% RSLogix 500 project PROJECT3.RSS, saved by version 8.40.00.08 %
PROJECT "UNTITLED"    % processor: Bul.1763 MicroLogix 1100 Series B %

PROGRAM FILES
  LAD 2   22 rungs

DATA FILES
  O0 OUTPUT  4 elements
  I1 INPUT  6 elements
  S2 STATUS  66 elements
  B3 BINARY  3 elements
  T4 TIMER  1 elements
  C5 COUNTER  1 elements
  R6 CONTROL  1 elements
  N7 INTEGER  18 elements
  F8 FLOAT  1 elements
  ST9   14 elements

LADDER 2
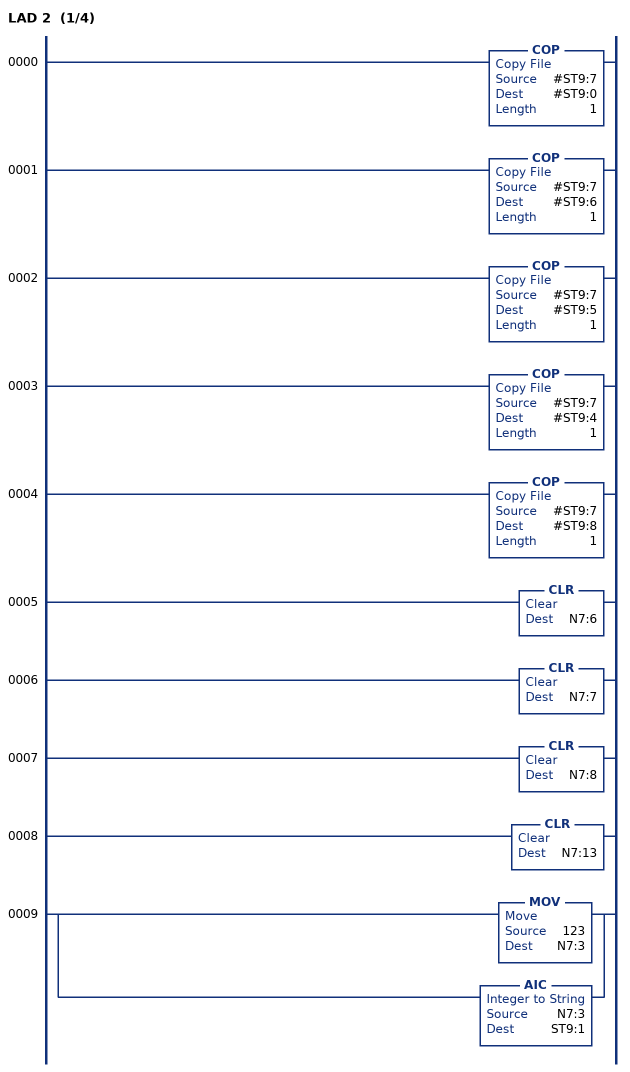
% Rung: 0 %
SOR COP #ST9:7 #ST9:0 1 EOR
% Rung: 1 %
SOR COP #ST9:7 #ST9:6 1 EOR
% Rung: 2 %
SOR COP #ST9:7 #ST9:5 1 EOR
% Rung: 3 %
SOR COP #ST9:7 #ST9:4 1 EOR
% Rung: 4 %
SOR COP #ST9:7 #ST9:8 1 EOR
% Rung: 5 %
SOR CLR N7:6 EOR
% Rung: 6 %
SOR CLR N7:7 EOR
% Rung: 7 %
SOR CLR N7:8 EOR
% Rung: 8 %
SOR CLR N7:13 EOR
% Rung: 9 %
SOR BST MOV 123 N7:3 NXB AIC N7:3 ST9:1 BND EOR

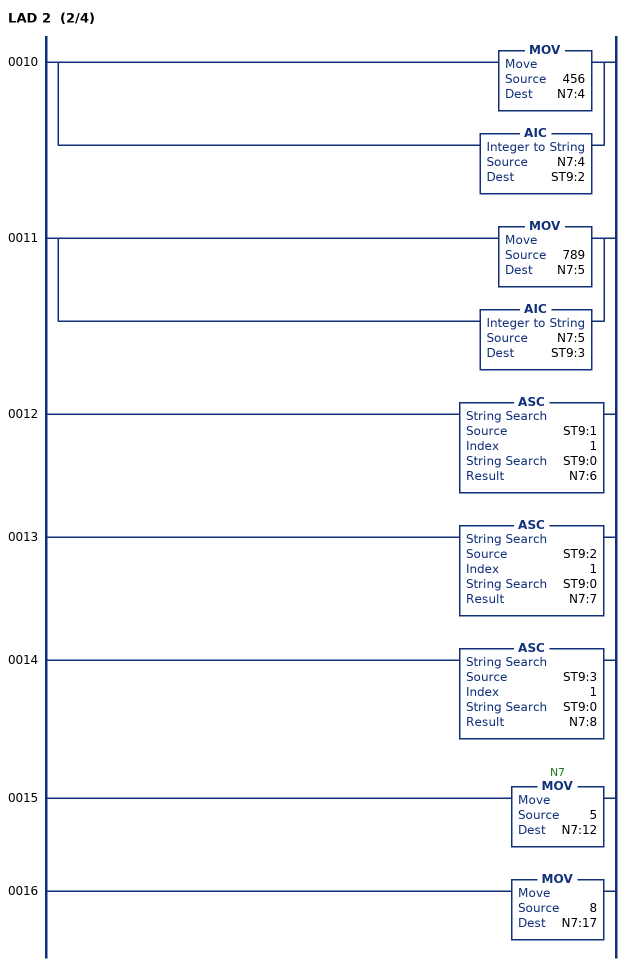
% Rung: 10 %
SOR BST MOV 456 N7:4 NXB AIC N7:4 ST9:2 BND EOR
% Rung: 11 %
SOR BST MOV 789 N7:5 NXB AIC N7:5 ST9:3 BND EOR
% Rung: 12 %
SOR ASC ST9:1 1 ST9:0 N7:6 EOR
% Rung: 13 %
SOR ASC ST9:2 1 ST9:0 N7:7 EOR
% Rung: 14 %
SOR ASC ST9:3 1 ST9:0 N7:8 EOR
% Rung: 15 %
SOR MOV 5 N7:12 EOR
%   N7:12  N7 %
% Rung: 16 %
SOR MOV 8 N7:17 EOR

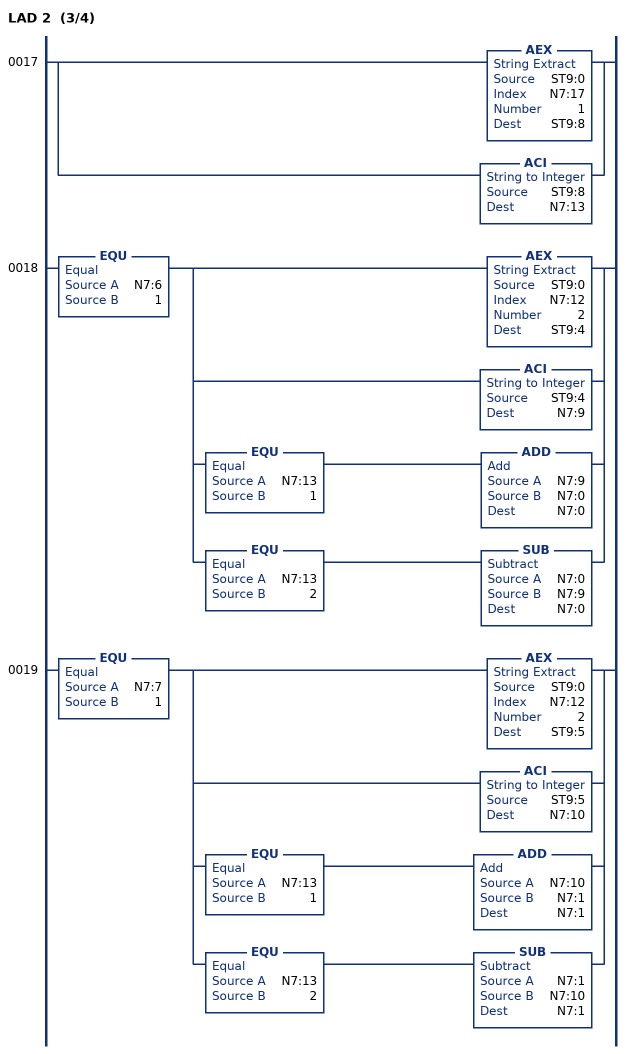
% Rung: 17 %
SOR BST AEX ST9:0 N7:17 1 ST9:8 NXB ACI ST9:8 N7:13 BND EOR
% Rung: 18 %
SOR EQU N7:6 1 BST AEX ST9:0 N7:12 2 ST9:4 NXB ACI ST9:4 N7:9 NXB EQU N7:13 1 ADD N7:9 N7:0 N7:0 NXB EQU N7:13 2 SUB N7:0 N7:9 N7:0 BND EOR
%   N7:12  N7 %
% Rung: 19 %
SOR EQU N7:7 1 BST AEX ST9:0 N7:12 2 ST9:5 NXB ACI ST9:5 N7:10 NXB EQU N7:13 1 ADD N7:10 N7:1 N7:1 NXB EQU N7:13 2 SUB N7:1 N7:10 N7:1 BND EOR
%   N7:12  N7 %

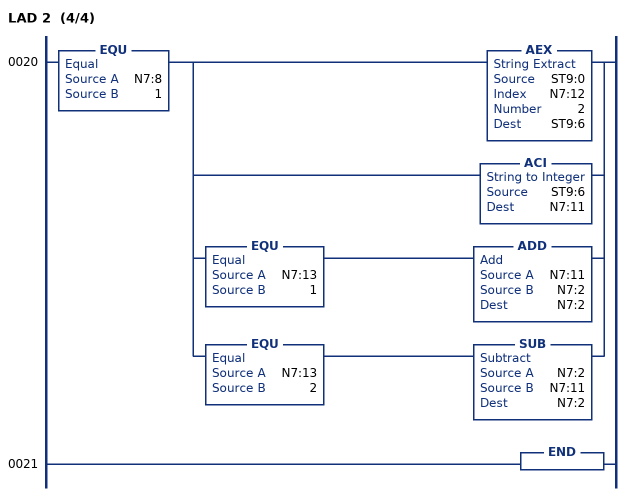
% Rung: 20 %
SOR EQU N7:8 1 BST AEX ST9:0 N7:12 2 ST9:6 NXB ACI ST9:6 N7:11 NXB EQU N7:13 1 ADD N7:11 N7:2 N7:2 NXB EQU N7:13 2 SUB N7:2 N7:11 N7:2 BND EOR
%   N7:12  N7 %
% Rung: 21 %
SOR END EOR

DATA TABLE (non-zero values as saved)
DATA N7
% N7:0 % 4 0 0 123 456 789 0 0 0 5
% N7:10 % 1 1 5 0 0 0 0 8
DATA ST9
% ST9:1 % "123"
% ST9:2 % "456"
% ST9:3 % "789"
